TYPE ST_ItemPK4_OUT3 :
STRUCT
	Identity		:ST_Identity_PK4_OUT3;
	ItemState		:STRING;
	RejectReason	:ST_RejectReason_PK4_OUT3;
	logs			:ST_logs_PK4_OUT3;
	NoRead			:STRING;
END_STRUCT
END_TYPE

(* stored: Version 1.1.0.1, ProductVersion 3.1.4024.13
   DUT ST_ItemPK4_OUT3: Id {f6ccc43a-61a9-4692-a2be-42c13c0447e0} *)
